# EPICS StreamDevice protocol: pfcu/protocols/pfcu.proto
Terminator = CR LF;

debugTest {
	Out "StreamDevice test success.";
#	Out 'ACQUIRE "%(\$1:testAI1)d";';
}

#insertPFCU {
#	out "!PFCU\$1 I%(1w1a:testAI1)d";
#}

#removePFCU {
#	out "!PFCU0%(\$1)d R%(A)d%(B)d%(C)d%(D)d";
#}

callPFCU {
	out "!PFCU03 I1234";
#	in  "\%PFCU03 OK 1234 DONE;";
	wait 500;
	out "!PFCU03 R%(\$1:PFCUmask.VAL)d";
}

InqFilPos {
    out "!PFCU03 P";
    in 0x25,0x50,0x46,0x43,0x55,0x30,0x33,0x20,0x4F,0x4B,0x20,0x20,"%b",0x20,"DONE;";
#   ExtraInput=Ignore;
}
